// xlh_base/app/IoT/DEVICES/_342_FB_DEVICE_Z2M_BATTERY_AQARA_SWITCH_H1
// =============================================================================
// _342_FB_DEVICE_Z2M_BATTERY_AQARA_SWITCH_H1
// -----------------------------------------------------------------------------
// Aqara H1 wireless wall switch — 2-button wireless switch with
// single/double/triple press detection (left, right, both simultaneously).
//
// Behavior of the boolean outputs:
//   - When an action is received, the corresponding output is set for
//     EXACTLY ONE PLC cycle (pulse). In the next cycle all outputs are
//     reset again — external logic can therefore work directly with
//     R_TRIG.
// =============================================================================
FUNCTION_BLOCK _342_FB_DEVICE_Z2M_BATTERY_AQARA_SWITCH_H1 EXTENDS _340_FB_DEVICE_Z2M_BATTERY
VAR_OUTPUT
    sAction       : STRING(255);    // Last reported action (diagnostics)
    bLeft         : BOOL;
    bLeftDouble   : BOOL;
    bLeftTriple   : BOOL;
    bRight        : BOOL;
    bRightDouble  : BOOL;
    bRightTriple  : BOOL;
    bBoth         : BOOL;
    bBothDouble   : BOOL;
    bBothTriple   : BOOL;
END_VAR
VAR
    _bNewAction : BOOL;     // TRUE in the cycle after an action has arrived
END_VAR

SUPER^();

IF _bNewAction THEN
    // One-cycle pulse on the matching output.
    _bNewAction  := FALSE;
    bLeft        := sAction = 'single_left';
    bLeftDouble  := sAction = 'double_left';
    bLeftTriple  := sAction = 'triple_left';
    bRight       := sAction = 'single_right';
    bRightDouble := sAction = 'double_right';
    bRightTriple := sAction = 'triple_right';
    bBoth        := sAction = 'single_both';
    bBothDouble  := sAction = 'double_both';
    bBothTriple  := sAction = 'triple_both';
ELSE
    bLeft        := FALSE;
    bLeftDouble  := FALSE;
    bLeftTriple  := FALSE;
    bRight       := FALSE;
    bRightDouble := FALSE;
    bRightTriple := FALSE;
    bBoth        := FALSE;
    bBothDouble  := FALSE;
    bBothTriple  := FALSE;
END_IF

// =============================================================================
// METHOD newMessage
// -----------------------------------------------------------------------------
// Reads the action from the event topic and triggers the pulse logic in
// the next cycle.
// =============================================================================
METHOD newMessage : BOOL
SUPER^.newMessage();
IF _fbMqttSubscriber.wsLastTopic = _wsMqttTopicEvent THEN
    sAction := GET_STRING_FROM_VALUE(sAction, GET_VALUE_FROM_MSG('action', ADR(_sSubscribedMessage)));
    THIS^._bNewAction := TRUE;
END_IF
END_METHOD

END_FUNCTION_BLOCK

// xlh_base/app/IoT/DEVICES/VISU/VISU_FB_DEVICE_SHELLY_RELAIS
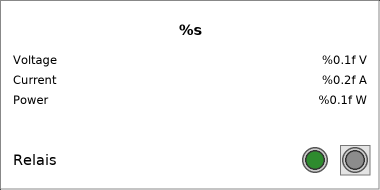
VISUALIZATION VISU_FB_DEVICE_SHELLY_RELAIS  // 380x190
VAR_INPUT
   {attribute 'parameterstringof' := 'fbDevice'}
   sFbInstanceName : STRING;
END_VAR
VAR_IN_OUT
   fbDevice: _201_FB_DEVICE_SHELLY_1PM_PLUG;
END_VAR
    Rectangle (0,0 381x191)
    Rectangle (10,140 281x40), "Relais"
    Rectangle (10,10 361x40), "%s", text variable: fbDevice.sLabel
    Lamp1 (300,140 30x40), variable: fbDevice.bRelaisState, style: Lamp-Lamp1-Green
    PushSwitch (340,140 30x40), variable: fbDevice.bRelais, behaviour: TOGGLE, style: Switch-PushSwitch-Gray
    Rectangle (10,50 261x20), "Voltage"
    Rectangle (270,50 100x20), "%0.1f V", text variable: fbDevice.fVoltage
    Rectangle (270,70 100x20), "%0.2f A", text variable: fbDevice.fCurrent
    Rectangle (10,70 261x20), "Current"
    Rectangle (270,90 100x20), "%0.1f W", text variable: fbDevice.fPower
    Rectangle (10,90 261x20), "Power"
END_VISUALIZATION

// xlh_base/app/VISUALIZATION
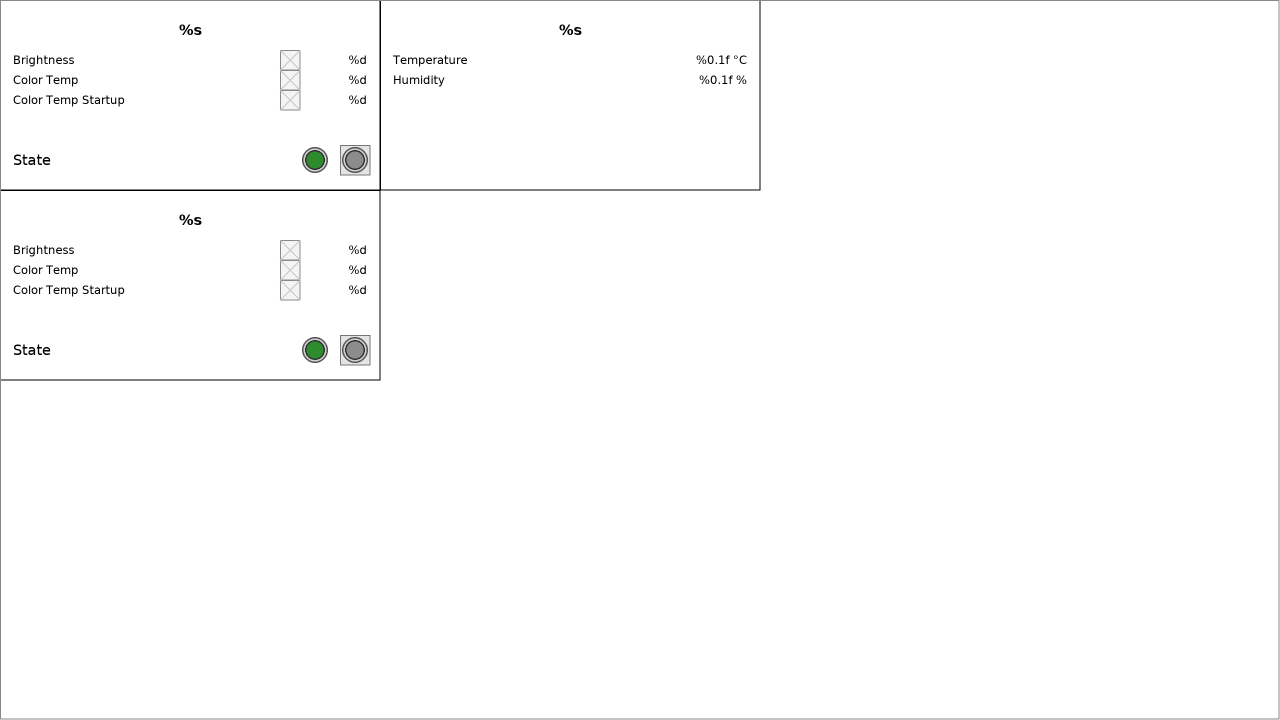
VISUALIZATION VISUALIZATION  // 1280x720
    Frame (0,0 380x191)
        shows _312_VISU_FB_DEVICE_Z2M_POWER_LAMP(fbDevice := io.fbLamp1)
    Frame (0,190 380x191)
        shows _312_VISU_FB_DEVICE_Z2M_POWER_LAMP(fbDevice := io.fbLamp2)
    Frame (380,0 380x191)
        shows _341_VISU_FB_DEVICE_Z2M_BATTERY_SONOFF_TEMP_HUM(fbDevice := io.fbTempHumSensor)
END_VISUALIZATION

// xlh_base/app/IoT/DEVICES/VISU/VISU_FB_DEVICE_SHELLY_RELAIS_TEMP
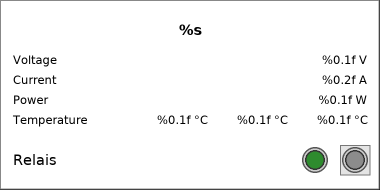
VISUALIZATION VISU_FB_DEVICE_SHELLY_RELAIS_TEMP  // 380x190
VAR_INPUT
   {attribute 'parameterstringof' := 'fbDevice'}
   sFbInstanceName : STRING;
END_VAR
VAR_IN_OUT
   fbDevice: _202_FB_DEVICE_SHELLY_1PM_TEMP;
END_VAR
    Rectangle (0,0 380x190)
    Rectangle (10,140 281x40), "Relais"
    Rectangle (10,10 361x40), "%s", text variable: fbDevice.sLabel
    Lamp1 (300,140 30x40), variable: fbDevice.bRelaisState, style: Lamp-Lamp1-Green
    PushSwitch (340,140 30x40), variable: fbDevice.bRelais, behaviour: TOGGLE, style: Switch-PushSwitch-Gray
    Rectangle (10,50 261x20), "Voltage"
    Rectangle (270,50 100x20), "%0.1f V", text variable: fbDevice.fVoltage
    Rectangle (270,70 100x20), "%0.2f A", text variable: fbDevice.fCurrent
    Rectangle (10,70 261x20), "Current"
    Rectangle (270,90 100x20), "%0.1f W", text variable: fbDevice.fPower
    Rectangle (10,90 261x20), "Power"
    Rectangle (10,110 111x20), "Temperature"
    Rectangle (210,110 81x20), "%0.1f °C", text variable: fbDevice.fTemperature2
    Rectangle (290,110 81x20), "%0.1f °C", text variable: fbDevice.fTemperature3
    Rectangle (130,110 81x20), "%0.1f °C", text variable: fbDevice.fTemperature1
END_VISUALIZATION

// xlh_base/app/IoT/DEVICES/VISU/_310_VISU_FB_DEVICE_Z2M_POWER_SWITCH
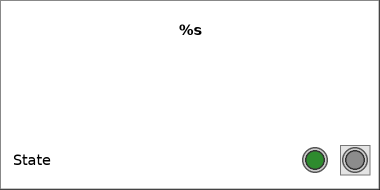
VISUALIZATION _310_VISU_FB_DEVICE_Z2M_POWER_SWITCH  // 380x190
VAR_INPUT
   {attribute 'parameterstringof' := 'fbDevice'}
   sFbInstanceName : STRING;
END_VAR
VAR_IN_OUT
   fbDevice: _310_FB_DEVICE_Z2M_POWER_SWITCH;
END_VAR
    Rectangle (0,0 380x190)
    Rectangle (10,140 281x40), "State"
    Rectangle (10,10 361x40), "%s", text variable: fbDevice.sLabel
    Lamp1 (300,140 30x40), variable: fbDevice.bOnState, style: Lamp-Lamp1-Green
    PushSwitch (340,140 30x40), variable: fbDevice.bOn, behaviour: TOGGLE, style: Switch-PushSwitch-Gray
END_VISUALIZATION

// xlh_base/app/IoT/DEVICES/VISU/_311_VISU_FB_DEVICE_Z2M_POWER_SWITCH_IKEAL_INSPELING
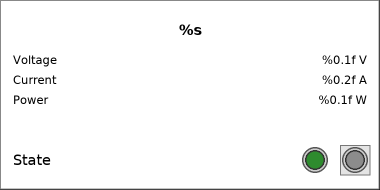
VISUALIZATION _311_VISU_FB_DEVICE_Z2M_POWER_SWITCH_IKEAL_INSPELING  // 380x190
VAR_INPUT
   {attribute 'parameterstringof' := 'fbDevice'}
   sFbInstanceName : STRING;
END_VAR
VAR_IN_OUT
   fbDevice: _311_FB_DEVICE_Z2M_POWER_SWITCH_IKEA_INSPELING;
END_VAR
    Rectangle (0,0 380x190)
    Rectangle (10,140 281x40), "State"
    Rectangle (10,10 361x40), "%s", text variable: fbDevice.sLabel
    Lamp1 (300,140 30x40), variable: fbDevice.bOnState, style: Lamp-Lamp1-Green
    PushSwitch (340,140 30x40), variable: fbDevice.bOn, behaviour: TOGGLE, style: Switch-PushSwitch-Gray
    Rectangle (270,50 100x20), "%0.1f V", text variable: fbDevice.fVoltage
    Rectangle (10,50 261x20), "Voltage"
    Rectangle (270,70 100x20), "%0.2f A", text variable: fbDevice.fCurrent
    Rectangle (10,70 261x20), "Current"
    Rectangle (270,90 100x20), "%0.1f W", text variable: fbDevice.fPower
    Rectangle (10,90 261x20), "Power"
END_VISUALIZATION

// xlh_base/app/IoT/DEVICES/VISU/_312_VISU_FB_DEVICE_Z2M_POWER_LAMP
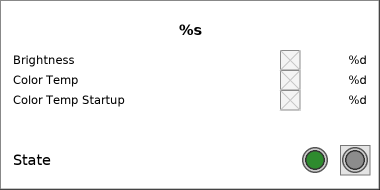
VISUALIZATION _312_VISU_FB_DEVICE_Z2M_POWER_LAMP  // 380x190
VAR_INPUT
   {attribute 'parameterstringof' := 'fbDevice'}
   sFbInstanceName : STRING;
END_VAR
VAR_IN_OUT
   fbDevice: _312_FB_DEVICE_Z2M_POWER_LAMP;
END_VAR
    Rectangle (0,0 380x190)
    Rectangle (10,140 281x40), "State"
    Rectangle (10,10 361x40), "%s", text variable: fbDevice.sLabel
    Lamp1 (300,140 30x40), variable: fbDevice.bOnState, style: Lamp-Lamp1-Green
    PushSwitch (340,140 30x40), variable: fbDevice.bOn, behaviour: TOGGLE, style: Switch-PushSwitch-Gray
    Rectangle (300,50 70x20), "%d", text variable: fbDevice.iBrightness
    Rectangle (10,50 261x20), "Brightness"
    Rectangle (300,70 70x20), "%d", text variable: fbDevice.iColorTemp
    Rectangle (10,70 261x20), "Color Temp"
    Rectangle (300,90 70x20), "%d", text variable: fbDevice.iColorTempStartup
    Rectangle (10,90 261x20), "Color Temp Startup"
    Image (280,50 20x20), invisible if: (fbDevice.iBrightness = -1) OR NOT fbDevice.bOnState, image: VisuSymbols.Symbols.Edit
        OnMouseClick: write fbDevice._iBrightnessWrite via Default, min 0, max 254
    Image (280,70 20x20), invisible if: (fbDevice.iColorTemp = -1) OR NOT fbDevice.bOnState, image: VisuSymbols.Symbols.Edit
        OnMouseClick: write fbDevice._iColorTempWrite via Default, min 250, max 454
    Image (280,90 20x20), invisible if: (fbDevice.iColorTempStartup = -1) OR NOT fbDevice.bOnState, image: VisuSymbols.Symbols.Edit
        OnMouseClick: write fbDevice._iColorTempStartupWrite via Default, min 250, max 454
END_VISUALIZATION

// xlh_base/app/IoT/DEVICES/VISU/_341_VISU_FB_DEVICE_Z2M_BATTERY_SONOFF_TEMP_HUM
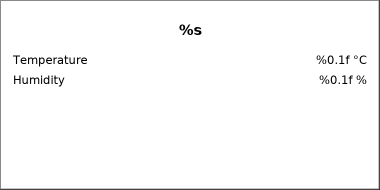
VISUALIZATION _341_VISU_FB_DEVICE_Z2M_BATTERY_SONOFF_TEMP_HUM  // 380x190
VAR_INPUT
   {attribute 'parameterstringof' := 'fbDevice'}
   sFbInstanceName : STRING;
END_VAR
VAR_IN_OUT
   fbDevice: _341_FB_DEVICE_Z2M_BATTERY_SONOFF_TEMP_HUM;
END_VAR
    Rectangle (0,0 380x190)
    Rectangle (10,10 361x40), "%s", text variable: fbDevice.sLabel
    Rectangle (300,50 70x20), "%0.1f °C", text variable: fbDevice.fTemperature
    Rectangle (10,50 261x20), "Temperature"
    Rectangle (300,70 70x20), "%0.1f %", text variable: fbDevice.fHumidity
    Rectangle (10,70 261x20), "Humidity"
END_VISUALIZATION
